FUNCTION_BLOCK EL3162
VAR
	_io : EL3xx2_Data;
	{attribute addProperty Name "WcState"}
	_wcState : WcStateInputToggle;
	{attribute addProperty Name "Info data"}
	_infoData : InfoDataAds;
END_VAR

PROPERTY IO : REFERENCE TO EL3xx2_Data
GET
IO REF= _io;
END_GET
END_PROPERTY

PROPERTY WcState : REFERENCE TO WcStateInputToggle
GET
WcState REF= _wcState;
END_GET
END_PROPERTY

END_FUNCTION_BLOCK

(* stored: Version 1.1.0.1, ProductVersion 3.1.4024.9
   POU EL3162: Id {a2104eba-eb55-0d55-3baf-84d28c6a9b02}, SpecialFunc None
   Property IO: Id {d197175a-1529-06bf-3c67-32dd531bf59e}
   Get Get: Id {04396854-7aad-043f-0849-c97c675c5b87}
   Property WcState: Id {20045e6c-daee-0f28-3f11-3aaab0ab7b17}
   Get Get: Id {848a3675-da5a-0255-019e-6165a9185a63} *)
